// TwinCAT 3 PLC project Motion_PLC_Practice
// ProgramVersion: 3.1.4023.0
// libraries:
//   lcls-twincat-motion, * (SLAC)
//   Tc2_Standard, * (Beckhoff Automation GmbH)
//   Tc2_System, * (Beckhoff Automation GmbH)
//   Tc3_Module, * (Beckhoff Automation GmbH)
// project tree:
//   / PlcTask.TcTTO
//   POUs/ MAIN.TcPOU
// real-time tasks:
//   TASK PlcTask: cycle T#10ms, priority 20, ADS port 350
// motion (NC):
//   TASK NC-Task 1 SAF: cycle T#2ms, priority 4, ADS port 501
//   TASK NC-Task 1 SVB: cycle T#10ms, priority 8, ADS port 511
//   AXIS Axis 1 (id 1)
//     Velo: Maximum=2
//     OtherSettings: AllowMotionCmdToSlave=true
//     encoder EncType=4
//       EncPara: MaxCount=#x0000ffff
//         Inc: RefSoftSyncMask=#x0000ffff
//     drive DrvType=24
//       Analog: VeloReferenz=1, TorqueSetpointScale=10, ScaleFactorActTorque=0.1
//       TimeComp: TaskDelayCycles=1
//     controller CtrType=1
//       CtrPara: PriorControlFactor=1
//         Observer: BandWidth=20
// I/O:
//   DEVICE Device 1 (EtherCAT), AmsNetId 172.21.148.87.2.1
//     Term 1 (EK1200) [EK1200-5000 EtherCAT Power supply (2A E-Bus)]
//       Term 2 (EL7031) [EL7031 1Ch. Stepper motor output stage (24V, 1.5A)]
//       Term 3 (EL1084) [EL1084 4Ch. Dig. Input 24V, 3ms, negative]
//       Term 4 (EL5042) [EL5042 2Ch. BiSS-C Encoder]
//       Term 5 (EL5021) [EL5021 1Ch. Sin/Cos Encoder]
//       Term 6 (EL9011) [EL9011 End Terminal]
// variable links:
//   NC-Task 1 SAF/Axes/Axis 1 <-> Device 1 (EtherCAT)/Term 1 (EK1200)/Term 2 (EL7031)
//     Drive/Inputs/In/nState1 @bit 3 <-> STM Status/Status/Error
//     Drive/Inputs/In/nState1 @bit 5 <-> STM Status/Status/Moving negative
//     Drive/Inputs/In/nState1 @bit 4 <-> STM Status/Status/Moving positive
//     Drive/Inputs/In/nState1 @bit 1 <-> STM Status/Status/Ready
//     Drive/Inputs/In/nState1 <-> STM Status/Status/Ready to enable
//     Drive/Inputs/In/nState1 @bit 6 <-> STM Status/Status/Torque reduced
//     Drive/Inputs/In/nState1 @bit 2 <-> STM Status/Status/Warning
//     Drive/Inputs/In/nState2 @bit 3 <-> STM Status/Status/Digital input 1
//     Drive/Inputs/In/nState2 @bit 4 <-> STM Status/Status/Digital input 2
//     Drive/Inputs/In/nState2 @bit 5 <-> STM Status/Status/Sync error
//     Drive/Inputs/In/nState2 @bit 7 <-> STM Status/Status/TxPDO Toggle
//     Drive/Inputs/In/nState4 @bit 1 <-> WcState/InputToggle
//     Drive/Inputs/In/nState4 <-> WcState/WcState
//     Drive/Outputs/Out/nCtrl1 <-> STM Control/Control/Enable
//     Drive/Outputs/Out/nCtrl1 @bit 2 <-> STM Control/Control/Reduce torque
//     Drive/Outputs/Out/nCtrl1 @bit 1 <-> STM Control/Control/Reset
//     Drive/Outputs/Out/nDataOut2[0] <-> STM Velocity/Velocity
//     Enc/Inputs/In/nDataIn1[0] <-> ENC Status compact/Counter value
//     Enc/Inputs/In/nDataIn2[0] <-> ENC Status compact/Latch value
//     Enc/Inputs/In/nState1 @bit 4 <-> ENC Status compact/Status/Counter overflow
//     Enc/Inputs/In/nState1 @bit 3 <-> ENC Status compact/Status/Counter underflow
//     Enc/Inputs/In/nState1 @bit 1 <-> ENC Status compact/Status/Latch extern valid
//     Enc/Inputs/In/nState1 @bit 2 <-> ENC Status compact/Status/Set counter done
//     Enc/Inputs/In/nState2 @bit 4 <-> ENC Status compact/Status/Status of extern latch
//     Enc/Inputs/In/nState2 @bit 5 <-> ENC Status compact/Status/Sync error
//     Enc/Inputs/In/nState2 @bit 7 <-> ENC Status compact/Status/TxPDO Toggle
//     Enc/Inputs/In/nState4 @bit 1 <-> WcState/InputToggle
//     Enc/Inputs/In/nState4 <-> WcState/WcState
//     Enc/Outputs/Out/nCtrl1 @bit 3 <-> ENC Control compact/Control/Enable latch extern on negative edge
//     Enc/Outputs/Out/nCtrl1 @bit 1 <-> ENC Control compact/Control/Enable latch extern on positive edge
//     Enc/Outputs/Out/nCtrl1 @bit 2 <-> ENC Control compact/Control/Set counter
//     Enc/Outputs/Out/nDataOut1[0] <-> ENC Control compact/Set counter value
//   Motion_PLC_Practice/Motion_PLC_Practice Instance <-> Device 1 (EtherCAT)/Term 1 (EK1200)/Term 3 (EL1084)
//     PlcTask Inputs/MAIN.backwardLimitSwitch <-> Channel 1/Input
//     PlcTask Inputs/MAIN.forwardLimitSwitch <-> Channel 2/Input
//   Motion_PLC_Practice/Motion_PLC_Practice Instance <-> Device 1 (EtherCAT)/Term 1 (EK1200)/Term 4 (EL5042)
//     PlcTask Inputs/MAIN.M1.nRawEncoderULINT <-> FB Inputs Channel 1/Position

CONFIGURATION Motion_PLC_Practice
    RESOURCE PLC ON TwinCAT3
        TASK PlcTask(INTERVAL := T#10ms, PRIORITY := 20);
        PROGRAM MAIN WITH PlcTask : MAIN;
    END_RESOURCE
END_CONFIGURATION

// ---- POUs/MAIN.TcPOU
PROGRAM MAIN
VAR
	// Define EPICS interface for moving motor (struct)
	{attribute 'TcLinkTo' := '.nRawEncoderULINT     := TIID^Device 1 (EtherCAT)^Term 1 (EK1200)^Term 4 (EL5042)^FB Inputs Channel 1^Position'}
	M1: ST_MotionStage := (sName := 'MOTION:PRACTICE',
                        bPowerSelf := True); // opt out of PMPS and handle
											// motor enabling within FB_MotionStage
	
	// Attribute Linking (for hardware)
	// Inputs (Limit Switch)
	{attribute 'TcLinkTo' := 'TIID^Device 1 (EtherCAT)^Term 1 (EK1200)^Term 3 (EL1084)^Channel 1^Input'}
	backwardLimitSwitch AT %I* : BOOL;
	
	{attribute 'TcLinkTo' := 'TIID^Device 1 (EtherCAT)^Term 1 (EK1200)^Term 3 (EL1084)^Channel 2^Input'}
	forwardLimitSwitch AT %I* : BOOL;
	
	// Function Block Logic 
	fbMotion1: FB_MotionStage;

END_VAR

// Limit switch is NPN, while motion library uses PNP
M1.bLimitForwardEnable := NOT forwardLimitSwitch;
M1.bLimitBackwardEnable := NOT backwardLimitSwitch;

M1.bHardwareEnable := TRUE; // ok to move

// Invoke function block call
fbMotion1(stMotionStage := M1);

END_PROGRAM
